(* CODESYS project wagolib787_01_twincat.library
   Company: Wago
   Title: T3_WagoLib787_01_TwinCat
   Placeholder: T3_WagoLib787_01_TwinCat
   Version: 1.0.0.0

Project tree, tasks and I/O mapping:
  libraries: Tc2_Standard, * (Beckhoff Automation GmbH); Tc2_System, * (Beckhoff Automation GmbH); Tc3_Interfaces, * (Beckhoff Automation GmbH); Tc3_Module, * (Beckhoff Automation GmbH)
  Data types/
    data type typEpsitronStatus
  Global Variables/
    global variables Global_Variables
    global variables Variable_Configuration
  POUs/
    function block FB787_1662 [ST]
    function block FB787_1662_ReadCurrent [ST]
    function block FB787_1664 [ST]
    function block FB787_1664_ReadCurrent [ST]
    function block FB787_1668 [ST]
    function block FB787_1668_ReadCurrent [ST]
    function FC787_Version [ST]
  Version/
    global variables Global_Version
  Visualizations/
*)

// Data types/typEpsitronStatus
TYPE typEpsitronStatus :
	(Ch_Active:=0,
	Ch_Warning:=1,
	Ch_Tripped:=2,
	Ch_not_Active:=3);
END_TYPE

// Global Variables/Global_Variables
{attribute 'Tc2GvlVarNames'}
VAR_GLOBAL
END_VAR

// Global Variables/Variable_Configuration
{attribute 'Tc2GvlVarNames'}
VAR_CONFIG
END_VAR

// Version/Global_Version
// This function has been automatically generated from the project information.
VAR_GLOBAL CONSTANT
	{attribute 'const_non_replaced'}
	{attribute 'linkalways'}
	stLibVersion_T3_WagoLib787_01_TwinCat : ST_LibVersion := (iMajor := 1, iMinor := 0, iBuild := 0, iRevision := 0, sVersion := '1.0.0.0');
END_VAR

// POUs/FB787_1662
FUNCTION_BLOCK FB787_1662
(***********************************************************************************************************	*)
(* Version: 1.0                                    			          														*)
(* Date: 05.09.2013                                   					          							            			*)
(***********************************************************************************************************	*)
(* WAGO Kontakttechnik GmbH Hansastr. 27 32423 Minden(Westf.)									*)
(* Tel. +0049 571/887-0 Fax. +0049 571/887-0															*)
(* Author: VB																								*)
(***********************************************************************************************************	*)
(*Description:	Epsitron electronic fuse (2 channel)	 													*)
(*Historie:																									*)
(*05.09.2013	VB		 Release																			*)
(***********************************************************************************************************	*)
VAR_INPUT
	xActive							:BOOL;
	xConfig						:BOOL;
	xChannel1Active				:BOOL;
	xChannel2Active				:BOOL;
	xS2_Input						:BOOL;
END_VAR
VAR_OUTPUT
	xDone							:BOOL;
	xConfigBusy					:BOOL;
	typChannel1Status			:typEpsitronStatus;(*0:Active,1:Warning,2:Tripped*)
	typChannel2Status			:typEpsitronStatus;
	xS1_Output					:BOOL;
END_VAR
VAR_IN_OUT
	xReset							:BOOL;
END_VAR
VAR
	a								: INT;
	state							: INT;
	TON1							: TON;
	aDaten						: ARRAY[0..44] OF BOOL;
	i								: INT;
	Ausgabe						: ARRAY[0..40] OF BOOL;
	go								: BOOL;
	init								: BOOL;
	R_TRIG1						: R_TRIG;
	auxExecute					: BOOL;
	xChannel3Active				:BOOL;
	xChannel4Active				:BOOL;
	xChannel5Active				: BOOL;
	xChannel6Active				: BOOL;
	xChannel7Active				: BOOL;
	xChannel8Active				: BOOL;
	auxReset						: BOOL;
END_VAR

IF xActive THEN
	R_TRIG1(CLK:=xConfig);
	IF r_trig1.q THEN
		auxExecute:=TRUE;
	END_IF
	
	CASE state OF
	0:(*ca. 1 Sekunde warten bis der Status abgefragt wird*)

		xS1_Output:=FALSE;
	
		IF NOT init THEN
			Ausgabe[0]:=1;
			Ausgabe[1]:=0;
			Ausgabe[2]:=1;
			Ausgabe[3]:=0;
			Ausgabe[4]:=1;
			Ausgabe[5]:=0;
			Ausgabe[6]:=1;
			Ausgabe[7]:=0;
			Ausgabe[8]:=1;
			Ausgabe[9]:=0;
			Ausgabe[10]:=1;
			Ausgabe[11]:=0;
			Ausgabe[12]:=1;
			Ausgabe[13]:=0;
			Ausgabe[14]:=1;
			Ausgabe[15]:=0;
			Ausgabe[16]:=1;
			Ausgabe[17]:=0;
			Ausgabe[18]:=1;
			Ausgabe[19]:=0;
			Ausgabe[20]:=1;
			Ausgabe[21]:=0;
			Ausgabe[22]:=1;
			Ausgabe[23]:=0;
			Ausgabe[24]:=1;
			Ausgabe[25]:=0;
			Ausgabe[26]:=1;
			Ausgabe[27]:=0;
			Ausgabe[28]:=1;
			Ausgabe[29]:=0;
			Ausgabe[30]:=1;
			Ausgabe[31]:=0;
			Ausgabe[32]:=1;
			Ausgabe[33]:=0;
			Ausgabe[34]:=0;
			Ausgabe[35]:=0;
			Ausgabe[36]:=0;
			Ausgabe[37]:=0;
			Ausgabe[38]:=0;
			Ausgabe[39]:=0;
			Ausgabe[40]:=0;
			init:=TRUE;
		END_IF

		IF auxExecute  THEN
			xConfigBusy:=TRUE;
			go:=TRUE;
			Ausgabe[0]:=1;
			Ausgabe[1]:=0;
			IF xChannel8Active THEN
				Ausgabe[2]:=0;
				Ausgabe[3]:=1;
			ELSE
				Ausgabe[2]:=1;
				Ausgabe[3]:=0;
			END_IF
		
			IF xChannel7Active THEN
				Ausgabe[4]:=0;
				Ausgabe[5]:=1;
			ELSE
				Ausgabe[4]:=1;
				Ausgabe[5]:=0;
			END_IF
			IF xChannel6Active THEN
				Ausgabe[6]:=0;
				Ausgabe[7]:=1;
			ELSE
				Ausgabe[6]:=1;
				Ausgabe[7]:=0;
			END_IF
			IF xChannel5Active THEN
				Ausgabe[8]:=0;
				Ausgabe[9]:=1;
			ELSE
				Ausgabe[8]:=1;
				Ausgabe[9]:=0;
			END_IF
			IF xChannel4Active THEN
				Ausgabe[10]:=0;
				Ausgabe[11]:=1;
			ELSE
				Ausgabe[10]:=1;
				Ausgabe[11]:=0;
			END_IF
			IF xChannel3Active THEN
				Ausgabe[12]:=0;
				Ausgabe[13]:=1;
			ELSE
				Ausgabe[12]:=1;
				Ausgabe[13]:=0;
			END_IF
			IF xChannel2Active THEN
				Ausgabe[14]:=0;
				Ausgabe[15]:=1;
			ELSE
				Ausgabe[14]:=1;
				Ausgabe[15]:=0;
			END_IF
			IF xChannel1Active THEN
				Ausgabe[16]:=0;
				Ausgabe[17]:=1;
			ELSE
				Ausgabe[16]:=1;
				Ausgabe[17]:=0;
			END_IF
			IF go THEN
				Ausgabe[18]:=0;
				Ausgabe[19]:=1;
			ELSE
				Ausgabe[18]:=1;
				Ausgabe[19]:=0;
			END_IF
				Ausgabe[20]:=1;
				Ausgabe[21]:=0;
				Ausgabe[22]:=1;
				Ausgabe[23]:=0;
				Ausgabe[24]:=1;
				Ausgabe[25]:=0;
				Ausgabe[26]:=1;
				Ausgabe[27]:=0;
				Ausgabe[28]:=1;
				Ausgabe[29]:=0;
				Ausgabe[30]:=1;
				Ausgabe[31]:=0;
				Ausgabe[32]:=1;
				Ausgabe[33]:=0;
				Ausgabe[34]:=0;
				Ausgabe[35]:=0;
				Ausgabe[36]:=0;
				Ausgabe[37]:=0;
				Ausgabe[38]:=0;
				Ausgabe[39]:=0;
				Ausgabe[40]:=0;
		END_IF;
	
		TON1(IN:=TRUE , PT:=t#1s);
		IF ton1.Q THEN
			state:=3;
			TON1(IN:=FALSE);
		END_IF


		(*Channel 1*)
		IF (aDaten[34] AND aDaten[35]) AND (aDaten[18] AND aDaten[19]) THEN
			typChannel1Status:=1;
		ELSIF (aDaten[34] AND aDaten[35]) AND (aDaten[18]=FALSE AND aDaten[19]=FALSE) THEN
			typChannel1Status:=2;
		ELSIF (aDaten[34]=FALSE AND aDaten[35]=FALSE) AND (aDaten[18]=FALSE AND aDaten[19]=FALSE) THEN
			typChannel1Status:=3;
		ELSE
			typChannel1Status:=0;
		END_IF

		(*Channel 2*)
		IF (aDaten[32] AND aDaten[33]) AND (aDaten[16] AND aDaten[17]) THEN
			typChannel2Status:=1;
		ELSIF (aDaten[32] AND aDaten[33]) AND (aDaten[16]=FALSE AND aDaten[17]=FALSE) THEN
			typChannel2Status:=2;
		ELSIF (aDaten[32]=FALSE AND aDaten[33]=FALSE) AND (aDaten[16]=FALSE AND aDaten[17]=FALSE) THEN
			typChannel2Status:=3;
		ELSE
			typChannel2Status:=0;
		END_IF


		IF auxReset AND xReset THEN
			xReset:=FALSE;
			auxReset:=FALSE;
		END_IF

	3:(*Reset Impuls mit 500ms ausführen*)
		IF xReset  THEN
			xS1_Output:=TRUE;
			TON1(IN:=TRUE , PT:=t#500ms);
			IF ton1.Q THEN
				state:=4;
				TON1(IN:=FALSE);
			END_IF
		ELSE
			state:=5;
			xS1_Output:=FALSE;
		END_IF
	
	4:(*Pause nach Reset*)
		TON1(IN:=TRUE , PT:=t#300ms);
		xS1_Output:=FALSE;
		IF ton1.Q THEN
			state:=5;
			TON1(IN:=FALSE);
			auxReset:=TRUE;
		END_IF

	5:
	(*Daten anfragen*)

		xS1_Output:=Ausgabe[a];
		aDaten[a+1]:=xS2_Input;
		a:=a+1;

		IF a>40 THEN
			state:=0;
			a:=0;
			i:=0;
			go:=FALSE;
			IF 	auxExecute AND xConfigBusy THEN(*schreibauftrag erledigt*)
				xDone:=FALSE;
				auxExecute:=FALSE;
				init:=FALSE;(*damit anschließend nur Daten ausgelesen werden. muss das Feld wieder den Lesecode bekommen*)
			ELSIF auxExecute AND NOT xConfigBusy THEN(*neuer  Schreibauftrag eingetroffen*)
				xConfigBusy:=TRUE;
				xDone:=FALSE;
			ELSE
				IF xConfig THEN
					xDone:=TRUE;
				ELSE
					xDone:=FALSE;
				END_IF
				xConfigBusy:=FALSE;
			END_IF
		ELSE
			;
		END_IF

	END_CASE
ELSE
	xS1_Output:=FALSE;
	state:=0;
	init:=0;
	a:=0;
	i:=0;
	auxReset:=FALSE;
END_IF

END_FUNCTION_BLOCK

// POUs/FB787_1662_ReadCurrent
FUNCTION_BLOCK FB787_1662_ReadCurrent
(***********************************************************************************************************	*)
(* Version: 1.0                                    			          														*)
(* Date: 05.09.2013                                   					          							            			*)
(***********************************************************************************************************	*)
(* WAGO Kontakttechnik GmbH Hansastr. 27 32423 Minden(Westf.)									*)
(* Tel. +0049 571/887-0 Fax. +0049 571/887-0															*)
(* Author: VB																								*)
(***********************************************************************************************************	*)
(*Description:	Epsitron electronic fuse with current overload protection	 							*)
(*Historie:																									*)
(*05.09.2013	VB		 			  																		*)
(***********************************************************************************************************	*)
VAR_INPUT
	xActive							:BOOL;
	xConfig						:BOOL;
	xChannel1Active				:BOOL;
	xChannel2Active				:BOOL;
	xReadSetting					:BOOL;(*0:read current,1:read setting*)
	xS2_Input						:BOOL;
END_VAR
VAR_OUTPUT
	xDone							:BOOL;
	xConfigBusy					:BOOL;
	typChannel1Status			:typEpsitronStatus;(*0:active,1:Überlast,2:Tripped,3:not_active*)
	typChannel2Status			:typEpsitronStatus;
	rVoltage						:REAL;
	rChannel1Current				:REAL;
	rChannel2Current				:REAL;
	iauxDisplay					:INT;
	xDisplaySettings				:BOOL;(*0:Channel value is current, 1:Channel value is setting*)
	xS1_Output					:BOOL;
END_VAR
VAR_IN_OUT
	xReset							:BOOL;
END_VAR
VAR
	xChannel3Active				:BOOL;
	xChannel4Active				:BOOL;
	xChannel5Active				:BOOL;
	xChannel6Active				:BOOL;
	xChannel7Active				:BOOL;
	xChannel8Active				:BOOL;
	typChannel3Status			:typEpsitronStatus;
	typChannel4Status			:typEpsitronStatus;
	typChannel5Status			:typEpsitronStatus;
	typChannel6Status			:typEpsitronStatus;
	typChannel7Status			:typEpsitronStatus;
	typChannel8Status			:typEpsitronStatus;
	rChannel3Current				:REAL;
	rChannel4Current				:REAL;
	rChannel5Current				:REAL;
	rChannel6Current				:REAL;
	rChannel7Current				:REAL;
	rChannel8Current				:REAL;
	a								: INT;
	state							: INT;
	TON1							: TON;
	aDaten						: ARRAY[0..188] OF BOOL;
	i								: INT;
	Ausgabe						: ARRAY[0..188] OF BOOL;
	go								: BOOL;
	init								: BOOL;
	R_TRIG1						: R_TRIG;
	auxExecute					: BOOL;
	auxReset						: BOOL;
	k								: INT;
	m								: INT;
	auxbyte						: BYTE;
	accurrentaux					: ARRAY[0..7]OF BYTE;
	bVoltage						: BYTE;
	auxProtocolBit5				: BOOL;
END_VAR

IF xActive THEN
	R_TRIG1(CLK:=xConfig);
	IF r_trig1.q THEN
		auxExecute:=TRUE;
	END_IF
	
	CASE state OF
	0:(*ca. 1 Sekunde warten bis der Status abgefragt wird*)

		xS1_Output:=FALSE;

		IF xReadSetting THEN
			Ausgabe[22]:=0;(*Bit 5->true*)
			Ausgabe[23]:=1;
		ELSE
			Ausgabe[22]:=1;
			Ausgabe[23]:=0;
		END_IF

		IF NOT init THEN
			FOR k:=0 TO 89 DO
				Ausgabe[2*k]:=1;
				Ausgabe[2*k+1]:=0;
			END_FOR
			FOR k:=0 TO 8 DO
				Ausgabe[178+k]:=0;
			END_FOR
			(*Protokoll 89 Bit*)
			Ausgabe[20]:=0;(*bit 6->true*)
			Ausgabe[21]:=1;

			IF xReadSetting THEN
				Ausgabe[22]:=0;(*Bit 5->true*)
				Ausgabe[23]:=1;
			ELSE
				Ausgabe[22]:=1;
				Ausgabe[23]:=0;
			END_IF

			init:=TRUE;
		END_IF

		IF auxExecute  THEN
			xConfigBusy:=TRUE;
			go:=TRUE;
			Ausgabe[0]:=1;
			Ausgabe[1]:=0;
			IF xChannel8Active THEN
				Ausgabe[2]:=0;
				Ausgabe[3]:=1;
			ELSE
				Ausgabe[2]:=1;
				Ausgabe[3]:=0;
			END_IF
		
			IF xChannel7Active THEN
				Ausgabe[4]:=0;
				Ausgabe[5]:=1;
			ELSE
				Ausgabe[4]:=1;
				Ausgabe[5]:=0;
			END_IF
			IF xChannel6Active THEN
				Ausgabe[6]:=0;
				Ausgabe[7]:=1;
			ELSE
				Ausgabe[6]:=1;
				Ausgabe[7]:=0;
			END_IF
			IF xChannel5Active THEN
				Ausgabe[8]:=0;
				Ausgabe[9]:=1;
			ELSE
				Ausgabe[8]:=1;
				Ausgabe[9]:=0;
			END_IF
			IF xChannel4Active THEN
				Ausgabe[10]:=0;
				Ausgabe[11]:=1;
			ELSE
				Ausgabe[10]:=1;
				Ausgabe[11]:=0;
			END_IF
			IF xChannel3Active THEN
				Ausgabe[12]:=0;
				Ausgabe[13]:=1;
			ELSE
				Ausgabe[12]:=1;
				Ausgabe[13]:=0;
			END_IF
			IF xChannel2Active THEN
				Ausgabe[14]:=0;
				Ausgabe[15]:=1;
			ELSE
				Ausgabe[14]:=1;
				Ausgabe[15]:=0;
			END_IF
			IF xChannel1Active THEN
				Ausgabe[16]:=0;
				Ausgabe[17]:=1;
			ELSE
				Ausgabe[16]:=1;
				Ausgabe[17]:=0;
			END_IF
			IF go THEN
				Ausgabe[18]:=0;
				Ausgabe[19]:=1;
			ELSE
				Ausgabe[18]:=1;
				Ausgabe[19]:=0;
			END_IF
			(*Protokoll 89 Bit*)
			Ausgabe[20]:=0;
			Ausgabe[21]:=1;
			IF xReadSetting THEN
				Ausgabe[22]:=0;(*Bit 5->true*)
				Ausgabe[23]:=1;
			ELSE
				Ausgabe[22]:=1;
				Ausgabe[23]:=0;
			END_IF

				FOR k:=0 TO 79 DO
					Ausgabe[24+2*k]:=1;
					Ausgabe[25+2*k]:=0;
				END_FOR

				Ausgabe[178]:=0;
				Ausgabe[179]:=0;
				Ausgabe[180]:=0;
				Ausgabe[181]:=0;
				Ausgabe[182]:=0;
				Ausgabe[183]:=0;
				Ausgabe[184]:=0;
				Ausgabe[185]:=0;
				Ausgabe[186]:=0;
				Ausgabe[187]:=0;
				Ausgabe[188]:=0;

		END_IF;

		TON1(IN:=TRUE , PT:=t#1s);
		IF ton1.Q THEN
			state:=3;
			TON1(IN:=FALSE);
		END_IF


		(*Channel 1*)
		IF (aDaten[34] (*AND aDaten[35]*)) AND (aDaten[18] AND aDaten[19]) THEN
			typChannel1Status:=1;
		ELSIF (aDaten[34] (*AND aDaten[35]*)) AND (aDaten[18]=FALSE AND aDaten[19]=FALSE) THEN
			typChannel1Status:=2;
		ELSIF (aDaten[34]=FALSE AND aDaten[35]=FALSE) AND (aDaten[18]=FALSE AND aDaten[19]=FALSE) THEN
			typChannel1Status:=3;
		ELSE
			typChannel1Status:=0;
		END_IF

		(*Channel 2*)
		IF (aDaten[32] AND aDaten[33]) AND (aDaten[16] AND aDaten[17]) THEN
			typChannel2Status:=1;
		ELSIF (aDaten[32] AND aDaten[33]) AND (aDaten[16]=FALSE AND aDaten[17]=FALSE) THEN
			typChannel2Status:=2;
		ELSIF (aDaten[32]=FALSE AND aDaten[33]=FALSE) AND (aDaten[16]=FALSE AND aDaten[17]=FALSE) THEN
			typChannel2Status:=3;
		ELSE
			typChannel2Status:=0;
		END_IF

		(*Channel 3*)
		IF (aDaten[30] AND aDaten[31]) AND (aDaten[14] AND aDaten[15]) THEN
			typChannel3Status:=1;
		ELSIF (aDaten[30] AND aDaten[31]) AND (aDaten[14]=FALSE AND aDaten[15]=FALSE) THEN
			typChannel3Status:=2;
		ELSIF (aDaten[30]=FALSE AND aDaten[31]=FALSE) AND (aDaten[14]=FALSE AND aDaten[15]=FALSE) THEN
			typChannel3Status:=3;
		ELSE
			typChannel3Status:=0;
		END_IF

		(*Channel 4*)
		IF (aDaten[28] AND aDaten[29]) AND (aDaten[12] AND aDaten[13]) THEN
			typChannel4Status:=1;
		ELSIF (aDaten[28] AND aDaten[29]) AND (aDaten[12]=FALSE AND aDaten[13]=FALSE) THEN
			typChannel4Status:=2;
		ELSIF (aDaten[28]=FALSE AND aDaten[29]=FALSE) AND (aDaten[12]=FALSE AND aDaten[13]=FALSE) THEN
			typChannel4Status:=3;
		ELSE
			typChannel4Status:=0;
		END_IF

	(*Channel 5*)
		IF (aDaten[26] AND aDaten[27]) AND (aDaten[10] AND aDaten[11]) THEN
			typChannel5Status:=1;
		ELSIF (aDaten[26] AND aDaten[27]) AND (aDaten[10]=FALSE AND aDaten[11]=FALSE) THEN
			typChannel5Status:=2;
		ELSIF (aDaten[26]=FALSE AND aDaten[27]=FALSE) AND (aDaten[10]=FALSE AND aDaten[11]=FALSE) THEN
			typChannel5Status:=3;
		ELSE
			typChannel5Status:=0;
		END_IF

	(*Channel 6*)
		IF (aDaten[24] AND aDaten[25]) AND (aDaten[8] AND aDaten[9]) THEN
			typChannel6Status:=1;
		ELSIF (aDaten[24] AND aDaten[25]) AND (aDaten[8]=FALSE AND aDaten[9]=FALSE) THEN
			typChannel6Status:=2;
		ELSIF (aDaten[24]=FALSE AND aDaten[25]=FALSE) AND (aDaten[8]=FALSE AND aDaten[9]=FALSE) THEN
			typChannel6Status:=3;
		ELSE
			typChannel6Status:=0;
		END_IF

	(*Channel 7*)
		IF (aDaten[22] AND aDaten[23]) AND (aDaten[6] AND aDaten[7]) THEN
			typChannel7Status:=1;
		ELSIF (aDaten[22] AND aDaten[23]) AND (aDaten[6]=FALSE AND aDaten[7]=FALSE) THEN
			typChannel7Status:=2;
		ELSIF (aDaten[22]=FALSE AND aDaten[23]=FALSE) AND (aDaten[6]=FALSE AND aDaten[7]=FALSE) THEN
			typChannel7Status:=3;
		ELSE
			typChannel7Status:=0;
		END_IF

	(*Channel 8*)
		IF (aDaten[20] AND aDaten[21]) AND (aDaten[4] AND aDaten[5]) THEN
			typChannel8Status:=1;
		ELSIF (aDaten[20] AND aDaten[21]) AND (aDaten[4]=FALSE AND aDaten[5]=FALSE) THEN
			typChannel8Status:=2;
		ELSIF (aDaten[20]=FALSE AND aDaten[21]=FALSE) AND (aDaten[4]=FALSE AND aDaten[5]=FALSE) THEN
			typChannel8Status:=3;
		ELSE
			typChannel8Status:=0;
		END_IF

		(*analog Werte Protokoll 89 bit*)
		IF (aDaten[36] AND aDaten[37]) THEN
			bVoltage.7:=TRUE;
		ELSE
			bVoltage.7:=FALSE;
		END_IF
		IF (aDaten[38] AND aDaten[39]) THEN
			bVoltage.6:=TRUE;
		ELSE
			bVoltage.6:=FALSE;
		END_IF
		IF (aDaten[40] AND aDaten[41]) THEN
			bVoltage.5:=TRUE;
		ELSE
			bVoltage.5:=FALSE;
		END_IF
		IF (aDaten[42] AND aDaten[43]) THEN
			bVoltage.4:=TRUE;
		ELSE
			bVoltage.4:=FALSE;
		END_IF
		IF (aDaten[44] AND aDaten[45]) THEN
			bVoltage.3:=TRUE;
		ELSE
			bVoltage.3:=FALSE;
		END_IF
		IF (aDaten[46] AND aDaten[47]) THEN
			bVoltage.2:=TRUE;
		ELSE
			bVoltage.2:=FALSE;
		END_IF
		IF (aDaten[48] AND aDaten[49]) THEN
			bVoltage.1:=TRUE;
		ELSE
			bVoltage.1:=FALSE;
		END_IF
		IF (aDaten[50] AND aDaten[51]) THEN
			bVoltage.0:=TRUE;
		ELSE
			bVoltage.0:=FALSE;
		END_IF
		IF bVoltage>0 THEN
			rVoltage:=BYTE_TO_REAL(bVoltage)/16+16;
		ELSE
			rVoltage:=0;
		END_IF

		FOR m:=0 TO 7 DO
			IF (aDaten[52+16*m] AND aDaten[53+16*m]) THEN
				auxbyte.7:=TRUE;
			ELSE
				auxbyte.7:=FALSE;
			END_IF
			IF (aDaten[54+16*m] AND aDaten[55+16*m]) THEN
				auxbyte.6:=TRUE;
			ELSE
				auxbyte.6:=FALSE;
			END_IF
			IF (aDaten[56+16*m] AND aDaten[57+16*m]) THEN
				auxbyte.5:=TRUE;
			ELSE
				auxbyte.5:=FALSE;
			END_IF
			IF (aDaten[58+16*m] AND aDaten[59+16*m]) THEN
				auxbyte.4:=TRUE;
			ELSE
				auxbyte.4:=FALSE;
			END_IF
			IF (aDaten[60+16*m] AND aDaten[61+16*m]) THEN
				auxbyte.3:=TRUE;
			ELSE
				auxbyte.3:=FALSE;
			END_IF
			IF (aDaten[62+16*m] AND aDaten[63+16*m]) THEN
				auxbyte.2:=TRUE;
			ELSE
				auxbyte.2:=FALSE;
			END_IF
			IF (aDaten[64+16*m] AND aDaten[65+16*m]) THEN
				auxbyte.1:=TRUE;
			ELSE
				auxbyte.1:=FALSE;
			END_IF
			IF (aDaten[66+16*m] AND aDaten[67+16*m]) THEN
				auxbyte.0:=TRUE;
			ELSE
				auxbyte.0:=FALSE;
			END_IF
			accurrentaux[m]:=auxbyte;
		END_FOR
		rChannel1Current:=BYTE_TO_REAL(accurrentaux[0])/16;
		rChannel2Current:=BYTE_TO_REAL(accurrentaux[1])/16;
		rChannel3Current:=BYTE_TO_REAL(accurrentaux[2])/16;
		rChannel4Current:=BYTE_TO_REAL(accurrentaux[3])/16;
		rChannel5Current:=BYTE_TO_REAL(accurrentaux[4])/16;
		rChannel6Current:=BYTE_TO_REAL(accurrentaux[5])/16;
		rChannel7Current:=BYTE_TO_REAL(accurrentaux[6])/16;
		rChannel8Current:=BYTE_TO_REAL(accurrentaux[7])/16;

		(*indicates wether current or setting values are displayed*)
		xDisplaySettings:=auxProtocolBit5;

		IF auxReset AND xReset THEN
			xReset:=FALSE;
			auxReset:=FALSE;
		END_IF

	3:(*Reset Impuls mit 500ms ausführen*)
		IF xReset  THEN
			xS1_Output:=TRUE;
			TON1(IN:=TRUE , PT:=t#500ms);
			IF ton1.Q THEN
				state:=4;
				TON1(IN:=FALSE);
			END_IF
		ELSE
			state:=5;
			xS1_Output:=FALSE;
		END_IF

	4:(*Pause nach Reset*)
		TON1(IN:=TRUE , PT:=t#300ms);
		xS1_Output:=FALSE;
		IF ton1.Q THEN
			state:=5;
			TON1(IN:=FALSE);
			auxReset:=TRUE;
		END_IF

	5:
	(*Daten anfragen*)

		xS1_Output:=Ausgabe[a];
		aDaten[a+1]:=xS2_Input;
		a:=a+1;
		iauxDisplay:=a;
		auxProtocolBit5:=NOT Ausgabe[22]; (*remember which values should be displayed->current or setting, dependen on bit5*)
		(*IF a>40 THEN*)
		IF a>184 THEN
			state:=0;
			a:=0;
			i:=0;
			go:=FALSE;
			IF 	auxExecute AND xConfigBusy THEN(*schreibauftrag erledigt*)
				xDone:=FALSE;
				auxExecute:=FALSE;
				init:=FALSE;(*damit anschließend nur Daten ausgelesen werden. muss das Feld wieder den Lesecode bekommen*)
			ELSIF auxExecute AND NOT xConfigBusy THEN(*neuer  Schreibauftrag eingetroffen*)
				xConfigBusy:=TRUE;
				xDone:=FALSE;
			ELSE
				IF xConfig THEN
					xDone:=TRUE;
				ELSE
					xDone:=FALSE;
				END_IF
				xConfigBusy:=FALSE;
			END_IF
		ELSE
			;
		END_IF

	END_CASE
ELSE
	xS1_Output:=FALSE;
	state:=0;
	init:=0;
	a:=0;
	i:=0;
	auxReset:=FALSE;
END_IF

END_FUNCTION_BLOCK

// POUs/FB787_1664
FUNCTION_BLOCK FB787_1664
(***********************************************************************************************************	*)
(* Version: 0.8                                    			          														*)
(* Date: 01.07.2012                                   					          							            			*)
(***********************************************************************************************************	*)
(* WAGO Kontakttechnik GmbH Hansastr. 27 32423 Minden(Westf.)									*)
(* Tel. +0049 571/887-0 Fax. +0049 571/887-0															*)
(* Author: VB																								*)
(***********************************************************************************************************	*)
(*Description:	Epsitron electronic fuse	 																*)
(*Historie:																									*)
(*01.07.2013	VB		 Version 0.8 changes according to FW2.00										*)
(*22.10.2012	VB		 Version 0.7 RC																	*)
(***********************************************************************************************************	*)
VAR_INPUT
	xActive							:BOOL;
	xConfig						:BOOL;
	xChannel1Active				:BOOL;
	xChannel2Active				:BOOL;
	xChannel3Active				:BOOL;
	xChannel4Active				:BOOL;
	xS2_Input						:BOOL;
END_VAR
VAR_OUTPUT
	xDone							:BOOL;
	xConfigBusy					:BOOL;
	typChannel1Status			:typEpsitronStatus;(*0:Active,1:Warning,2:Tripped*)
	typChannel2Status			:typEpsitronStatus;
	typChannel3Status			:typEpsitronStatus;
	typChannel4Status			:typEpsitronStatus;
	xS1_Output					:BOOL;
END_VAR
VAR_IN_OUT
	xReset							:BOOL;
END_VAR
VAR
	a								: INT;
	state							: INT;
	TON1							: TON;
	aDaten						: ARRAY[0..44] OF BOOL;
	i								: INT;
	Ausgabe						: ARRAY[0..40] OF BOOL;
	go								: BOOL;
	init								: BOOL;
	R_TRIG1						: R_TRIG;
	auxExecute					: BOOL;
	xChannel5Active				: BOOL;
	xChannel6Active				: BOOL;
	xChannel7Active				: BOOL;
	xChannel8Active				: BOOL;
	auxReset						: BOOL;
END_VAR

IF xActive THEN
	R_TRIG1(CLK:=xConfig);
	IF r_trig1.q THEN
		auxExecute:=TRUE;
	END_IF
	
	CASE state OF
	0:(*ca. 1 Sekunde warten bis der Status abgefragt wird*)

		xS1_Output:=FALSE;
	
		IF NOT init THEN
			Ausgabe[0]:=1;
			Ausgabe[1]:=0;
			Ausgabe[2]:=1;
			Ausgabe[3]:=0;
			Ausgabe[4]:=1;
			Ausgabe[5]:=0;
			Ausgabe[6]:=1;
			Ausgabe[7]:=0;
			Ausgabe[8]:=1;
			Ausgabe[9]:=0;
			Ausgabe[10]:=1;
			Ausgabe[11]:=0;
			Ausgabe[12]:=1;
			Ausgabe[13]:=0;
			Ausgabe[14]:=1;
			Ausgabe[15]:=0;
			Ausgabe[16]:=1;
			Ausgabe[17]:=0;
			Ausgabe[18]:=1;
			Ausgabe[19]:=0;
			Ausgabe[20]:=1;
			Ausgabe[21]:=0;
			Ausgabe[22]:=1;
			Ausgabe[23]:=0;
			Ausgabe[24]:=1;
			Ausgabe[25]:=0;
			Ausgabe[26]:=1;
			Ausgabe[27]:=0;
			Ausgabe[28]:=1;
			Ausgabe[29]:=0;
			Ausgabe[30]:=1;
			Ausgabe[31]:=0;
			Ausgabe[32]:=1;
			Ausgabe[33]:=0;
			Ausgabe[34]:=0;
			Ausgabe[35]:=0;
			Ausgabe[36]:=0;
			Ausgabe[37]:=0;
			Ausgabe[38]:=0;
			Ausgabe[39]:=0;
			Ausgabe[40]:=0;
			init:=TRUE;
		END_IF

		IF auxExecute  THEN
			xConfigBusy:=TRUE;
			go:=TRUE;
			Ausgabe[0]:=1;
			Ausgabe[1]:=0;
			IF xChannel8Active THEN
				Ausgabe[2]:=0;
				Ausgabe[3]:=1;
			ELSE
				Ausgabe[2]:=1;
				Ausgabe[3]:=0;
			END_IF
		
			IF xChannel7Active THEN
				Ausgabe[4]:=0;
				Ausgabe[5]:=1;
			ELSE
				Ausgabe[4]:=1;
				Ausgabe[5]:=0;
			END_IF
			IF xChannel6Active THEN
				Ausgabe[6]:=0;
				Ausgabe[7]:=1;
			ELSE
				Ausgabe[6]:=1;
				Ausgabe[7]:=0;
			END_IF
			IF xChannel5Active THEN
				Ausgabe[8]:=0;
				Ausgabe[9]:=1;
			ELSE
				Ausgabe[8]:=1;
				Ausgabe[9]:=0;
			END_IF
			IF xChannel4Active THEN
				Ausgabe[10]:=0;
				Ausgabe[11]:=1;
			ELSE
				Ausgabe[10]:=1;
				Ausgabe[11]:=0;
			END_IF
			IF xChannel3Active THEN
				Ausgabe[12]:=0;
				Ausgabe[13]:=1;
			ELSE
				Ausgabe[12]:=1;
				Ausgabe[13]:=0;
			END_IF
			IF xChannel2Active THEN
				Ausgabe[14]:=0;
				Ausgabe[15]:=1;
			ELSE
				Ausgabe[14]:=1;
				Ausgabe[15]:=0;
			END_IF
			IF xChannel1Active THEN
				Ausgabe[16]:=0;
				Ausgabe[17]:=1;
			ELSE
				Ausgabe[16]:=1;
				Ausgabe[17]:=0;
			END_IF
			IF go THEN
				Ausgabe[18]:=0;
				Ausgabe[19]:=1;
			ELSE
				Ausgabe[18]:=1;
				Ausgabe[19]:=0;
			END_IF
				Ausgabe[20]:=1;
				Ausgabe[21]:=0;
				Ausgabe[22]:=1;
				Ausgabe[23]:=0;
				Ausgabe[24]:=1;
				Ausgabe[25]:=0;
				Ausgabe[26]:=1;
				Ausgabe[27]:=0;
				Ausgabe[28]:=1;
				Ausgabe[29]:=0;
				Ausgabe[30]:=1;
				Ausgabe[31]:=0;
				Ausgabe[32]:=1;
				Ausgabe[33]:=0;
				Ausgabe[34]:=0;
				Ausgabe[35]:=0;
				Ausgabe[36]:=0;
				Ausgabe[37]:=0;
				Ausgabe[38]:=0;
				Ausgabe[39]:=0;
				Ausgabe[40]:=0;
		END_IF;
	
		TON1(IN:=TRUE , PT:=t#1s);
		IF ton1.Q THEN
			state:=3;
			TON1(IN:=FALSE);
		END_IF


		(*Channel 1*)
		IF (aDaten[34] AND aDaten[35]) AND (aDaten[18] AND aDaten[19]) THEN
			typChannel1Status:=1;
		ELSIF (aDaten[34] AND aDaten[35]) AND (aDaten[18]=FALSE AND aDaten[19]=FALSE) THEN
			typChannel1Status:=2;
		ELSIF (aDaten[34]=FALSE AND aDaten[35]=FALSE) AND (aDaten[18]=FALSE AND aDaten[19]=FALSE) THEN
			typChannel1Status:=3;
		ELSE
			typChannel1Status:=0;
		END_IF

		(*Channel 2*)
		IF (aDaten[32] AND aDaten[33]) AND (aDaten[16] AND aDaten[17]) THEN
			typChannel2Status:=1;
		ELSIF (aDaten[32] AND aDaten[33]) AND (aDaten[16]=FALSE AND aDaten[17]=FALSE) THEN
			typChannel2Status:=2;
		ELSIF (aDaten[32]=FALSE AND aDaten[33]=FALSE) AND (aDaten[16]=FALSE AND aDaten[17]=FALSE) THEN
			typChannel2Status:=3;
		ELSE
			typChannel2Status:=0;
		END_IF

		(*Channel 3*)
		IF (aDaten[30] AND aDaten[31]) AND (aDaten[14] AND aDaten[15]) THEN
			typChannel3Status:=1;
		ELSIF (aDaten[30] AND aDaten[31]) AND (aDaten[14]=FALSE AND aDaten[15]=FALSE) THEN
			typChannel3Status:=2;
		ELSIF (aDaten[30]=FALSE AND aDaten[31]=FALSE) AND (aDaten[14]=FALSE AND aDaten[15]=FALSE) THEN
			typChannel3Status:=3;
		ELSE
			typChannel3Status:=0;
		END_IF

		(*Channel 4*)
		IF (aDaten[28] AND aDaten[29]) AND (aDaten[12] AND aDaten[13]) THEN
			typChannel4Status:=1;
		ELSIF (aDaten[28] AND aDaten[29]) AND (aDaten[12]=FALSE AND aDaten[13]=FALSE) THEN
			typChannel4Status:=2;
		ELSIF (aDaten[28]=FALSE AND aDaten[29]=FALSE) AND (aDaten[12]=FALSE AND aDaten[13]=FALSE) THEN
			typChannel4Status:=3;
		ELSE
			typChannel4Status:=0;
		END_IF



		IF auxReset AND xReset THEN
			xReset:=FALSE;
			auxReset:=FALSE;
		END_IF

	3:(*Reset Impuls mit 500ms ausführen*)
		IF xReset  THEN
			xS1_Output:=TRUE;
			TON1(IN:=TRUE , PT:=t#500ms);
			IF ton1.Q THEN
				state:=4;
				TON1(IN:=FALSE);
			END_IF
		ELSE
			state:=5;
			xS1_Output:=FALSE;
		END_IF
	
	4:(*Pause nach Reset*)
		TON1(IN:=TRUE , PT:=t#300ms);
		xS1_Output:=FALSE;
		IF ton1.Q THEN
			state:=5;
			TON1(IN:=FALSE);
			auxReset:=TRUE;
		END_IF

	5:
	(*Daten anfragen*)

		xS1_Output:=Ausgabe[a];
		aDaten[a+1]:=xS2_Input;
		a:=a+1;

		IF a>40 THEN
			state:=0;
			a:=0;
			i:=0;
			go:=FALSE;
			IF 	auxExecute AND xConfigBusy THEN(*schreibauftrag erledigt*)
				xDone:=FALSE;
				auxExecute:=FALSE;
				init:=FALSE;(*damit anschließend nur Daten ausgelesen werden. muss das Feld wieder den Lesecode bekommen*)
			ELSIF auxExecute AND NOT xConfigBusy THEN(*neuer  Schreibauftrag eingetroffen*)
				xConfigBusy:=TRUE;
				xDone:=FALSE;
			ELSE
				IF xConfig THEN
					xDone:=TRUE;
				ELSE
					xDone:=FALSE;
				END_IF
				xConfigBusy:=FALSE;
			END_IF
		ELSE
			;
		END_IF

	END_CASE
ELSE
	xS1_Output:=FALSE;
	state:=0;
	init:=0;
	a:=0;
	i:=0;
	auxReset:=FALSE;
END_IF

END_FUNCTION_BLOCK

// POUs/FB787_1664_ReadCurrent
FUNCTION_BLOCK FB787_1664_ReadCurrent
(***********************************************************************************************************	*)
(* Version: 1.0                                    			          														*)
(* Date: 05.09.2013                                   					          							            			*)
(***********************************************************************************************************	*)
(* WAGO Kontakttechnik GmbH Hansastr. 27 32423 Minden(Westf.)									*)
(* Tel. +0049 571/887-0 Fax. +0049 571/887-0															*)
(* Author: VB																								*)
(***********************************************************************************************************	*)
(*Description:	Epsitron electronic fuse with current overload protection	 							*)
(*Historie:																									*)
(*05.09.2013	VB		 			released  																*)
(***********************************************************************************************************	*)
VAR_INPUT
	xActive							:BOOL;
	xConfig						:BOOL;
	xChannel1Active				:BOOL;
	xChannel2Active				:BOOL;
	xChannel3Active				:BOOL;
	xChannel4Active				:BOOL;
	xReadSetting					:BOOL;(*0:read current,1:read setting*)
	xS2_Input						:BOOL;
END_VAR
VAR_OUTPUT
	xDone							:BOOL;
	xConfigBusy					:BOOL;
	typChannel1Status			:typEpsitronStatus;(*0:active,1:Überlast,2:Tripped,3:not_active*)
	typChannel2Status			:typEpsitronStatus;
	typChannel3Status			:typEpsitronStatus;
	typChannel4Status			:typEpsitronStatus;
	rVoltage						:REAL;
	rChannel1Current				:REAL;
	rChannel2Current				:REAL;
	rChannel3Current				:REAL;
	rChannel4Current				:REAL;
	iauxDisplay					:INT;
	xDisplaySettings				:BOOL;(*0:Channel value is current, 1:Channel value is setting*)
	xS1_Output					:BOOL;
END_VAR
VAR_IN_OUT
	xReset							:BOOL;
END_VAR
VAR
	xChannel5Active				:BOOL;
	xChannel6Active				:BOOL;
	xChannel7Active				:BOOL;
	xChannel8Active				:BOOL;
	typChannel5Status			:typEpsitronStatus;
	typChannel6Status			:typEpsitronStatus;
	typChannel7Status			:typEpsitronStatus;
	typChannel8Status			:typEpsitronStatus;
	rChannel5Current				:REAL;
	rChannel6Current				:REAL;
	rChannel7Current				:REAL;
	rChannel8Current				:REAL;
	a								: INT;
	state							: INT;
	TON1							: TON;
	aDaten						: ARRAY[0..188] OF BOOL;
	i								: INT;
	Ausgabe						: ARRAY[0..188] OF BOOL;
	go								: BOOL;
	init								: BOOL;
	R_TRIG1						: R_TRIG;
	auxExecute					: BOOL;
	auxReset						: BOOL;
	k								: INT;
	m								: INT;
	auxbyte						: BYTE;
	accurrentaux					: ARRAY[0..7]OF BYTE;
	bVoltage						: BYTE;
	auxProtocolBit5				: BOOL;
END_VAR

IF xActive THEN
	R_TRIG1(CLK:=xConfig);
	IF r_trig1.q THEN
		auxExecute:=TRUE;
	END_IF
	
	CASE state OF
	0:(*ca. 1 Sekunde warten bis der Status abgefragt wird*)

		xS1_Output:=FALSE;

		IF xReadSetting THEN
			Ausgabe[22]:=0;(*Bit 5->true*)
			Ausgabe[23]:=1;
		ELSE
			Ausgabe[22]:=1;
			Ausgabe[23]:=0;
		END_IF

		IF NOT init THEN
			FOR k:=0 TO 89 DO
				Ausgabe[2*k]:=1;
				Ausgabe[2*k+1]:=0;
			END_FOR
			FOR k:=0 TO 8 DO
				Ausgabe[178+k]:=0;
			END_FOR
			(*Protokoll 89 Bit*)
			Ausgabe[20]:=0;(*bit 6->true*)
			Ausgabe[21]:=1;

			IF xReadSetting THEN
				Ausgabe[22]:=0;(*Bit 5->true*)
				Ausgabe[23]:=1;
			ELSE
				Ausgabe[22]:=1;
				Ausgabe[23]:=0;
			END_IF

			init:=TRUE;
		END_IF

		IF auxExecute  THEN
			xConfigBusy:=TRUE;
			go:=TRUE;
			Ausgabe[0]:=1;
			Ausgabe[1]:=0;
			IF xChannel8Active THEN
				Ausgabe[2]:=0;
				Ausgabe[3]:=1;
			ELSE
				Ausgabe[2]:=1;
				Ausgabe[3]:=0;
			END_IF
		
			IF xChannel7Active THEN
				Ausgabe[4]:=0;
				Ausgabe[5]:=1;
			ELSE
				Ausgabe[4]:=1;
				Ausgabe[5]:=0;
			END_IF
			IF xChannel6Active THEN
				Ausgabe[6]:=0;
				Ausgabe[7]:=1;
			ELSE
				Ausgabe[6]:=1;
				Ausgabe[7]:=0;
			END_IF
			IF xChannel5Active THEN
				Ausgabe[8]:=0;
				Ausgabe[9]:=1;
			ELSE
				Ausgabe[8]:=1;
				Ausgabe[9]:=0;
			END_IF
			IF xChannel4Active THEN
				Ausgabe[10]:=0;
				Ausgabe[11]:=1;
			ELSE
				Ausgabe[10]:=1;
				Ausgabe[11]:=0;
			END_IF
			IF xChannel3Active THEN
				Ausgabe[12]:=0;
				Ausgabe[13]:=1;
			ELSE
				Ausgabe[12]:=1;
				Ausgabe[13]:=0;
			END_IF
			IF xChannel2Active THEN
				Ausgabe[14]:=0;
				Ausgabe[15]:=1;
			ELSE
				Ausgabe[14]:=1;
				Ausgabe[15]:=0;
			END_IF
			IF xChannel1Active THEN
				Ausgabe[16]:=0;
				Ausgabe[17]:=1;
			ELSE
				Ausgabe[16]:=1;
				Ausgabe[17]:=0;
			END_IF
			IF go THEN
				Ausgabe[18]:=0;
				Ausgabe[19]:=1;
			ELSE
				Ausgabe[18]:=1;
				Ausgabe[19]:=0;
			END_IF
			(*Protokoll 89 Bit*)
			Ausgabe[20]:=0;
			Ausgabe[21]:=1;
			IF xReadSetting THEN
				Ausgabe[22]:=0;(*Bit 5->true*)
				Ausgabe[23]:=1;
			ELSE
				Ausgabe[22]:=1;
				Ausgabe[23]:=0;
			END_IF

				FOR k:=0 TO 79 DO
					Ausgabe[24+2*k]:=1;
					Ausgabe[25+2*k]:=0;
				END_FOR

				Ausgabe[178]:=0;
				Ausgabe[179]:=0;
				Ausgabe[180]:=0;
				Ausgabe[181]:=0;
				Ausgabe[182]:=0;
				Ausgabe[183]:=0;
				Ausgabe[184]:=0;
				Ausgabe[185]:=0;
				Ausgabe[186]:=0;
				Ausgabe[187]:=0;
				Ausgabe[188]:=0;

		END_IF;

		TON1(IN:=TRUE , PT:=t#1s);
		IF ton1.Q THEN
			state:=3;
			TON1(IN:=FALSE);
		END_IF


		(*Channel 1*)
		IF (aDaten[34] (*AND aDaten[35]*)) AND (aDaten[18] AND aDaten[19]) THEN
			typChannel1Status:=1;
		ELSIF (aDaten[34] (*AND aDaten[35]*)) AND (aDaten[18]=FALSE AND aDaten[19]=FALSE) THEN
			typChannel1Status:=2;
		ELSIF (aDaten[34]=FALSE AND aDaten[35]=FALSE) AND (aDaten[18]=FALSE AND aDaten[19]=FALSE) THEN
			typChannel1Status:=3;
		ELSE
			typChannel1Status:=0;
		END_IF

		(*Channel 2*)
		IF (aDaten[32] AND aDaten[33]) AND (aDaten[16] AND aDaten[17]) THEN
			typChannel2Status:=1;
		ELSIF (aDaten[32] AND aDaten[33]) AND (aDaten[16]=FALSE AND aDaten[17]=FALSE) THEN
			typChannel2Status:=2;
		ELSIF (aDaten[32]=FALSE AND aDaten[33]=FALSE) AND (aDaten[16]=FALSE AND aDaten[17]=FALSE) THEN
			typChannel2Status:=3;
		ELSE
			typChannel2Status:=0;
		END_IF

		(*Channel 3*)
		IF (aDaten[30] AND aDaten[31]) AND (aDaten[14] AND aDaten[15]) THEN
			typChannel3Status:=1;
		ELSIF (aDaten[30] AND aDaten[31]) AND (aDaten[14]=FALSE AND aDaten[15]=FALSE) THEN
			typChannel3Status:=2;
		ELSIF (aDaten[30]=FALSE AND aDaten[31]=FALSE) AND (aDaten[14]=FALSE AND aDaten[15]=FALSE) THEN
			typChannel3Status:=3;
		ELSE
			typChannel3Status:=0;
		END_IF

		(*Channel 4*)
		IF (aDaten[28] AND aDaten[29]) AND (aDaten[12] AND aDaten[13]) THEN
			typChannel4Status:=1;
		ELSIF (aDaten[28] AND aDaten[29]) AND (aDaten[12]=FALSE AND aDaten[13]=FALSE) THEN
			typChannel4Status:=2;
		ELSIF (aDaten[28]=FALSE AND aDaten[29]=FALSE) AND (aDaten[12]=FALSE AND aDaten[13]=FALSE) THEN
			typChannel4Status:=3;
		ELSE
			typChannel4Status:=0;
		END_IF

	(*Channel 5*)
		IF (aDaten[26] AND aDaten[27]) AND (aDaten[10] AND aDaten[11]) THEN
			typChannel5Status:=1;
		ELSIF (aDaten[26] AND aDaten[27]) AND (aDaten[10]=FALSE AND aDaten[11]=FALSE) THEN
			typChannel5Status:=2;
		ELSIF (aDaten[26]=FALSE AND aDaten[27]=FALSE) AND (aDaten[10]=FALSE AND aDaten[11]=FALSE) THEN
			typChannel5Status:=3;
		ELSE
			typChannel5Status:=0;
		END_IF

	(*Channel 6*)
		IF (aDaten[24] AND aDaten[25]) AND (aDaten[8] AND aDaten[9]) THEN
			typChannel6Status:=1;
		ELSIF (aDaten[24] AND aDaten[25]) AND (aDaten[8]=FALSE AND aDaten[9]=FALSE) THEN
			typChannel6Status:=2;
		ELSIF (aDaten[24]=FALSE AND aDaten[25]=FALSE) AND (aDaten[8]=FALSE AND aDaten[9]=FALSE) THEN
			typChannel6Status:=3;
		ELSE
			typChannel6Status:=0;
		END_IF

	(*Channel 7*)
		IF (aDaten[22] AND aDaten[23]) AND (aDaten[6] AND aDaten[7]) THEN
			typChannel7Status:=1;
		ELSIF (aDaten[22] AND aDaten[23]) AND (aDaten[6]=FALSE AND aDaten[7]=FALSE) THEN
			typChannel7Status:=2;
		ELSIF (aDaten[22]=FALSE AND aDaten[23]=FALSE) AND (aDaten[6]=FALSE AND aDaten[7]=FALSE) THEN
			typChannel7Status:=3;
		ELSE
			typChannel7Status:=0;
		END_IF

	(*Channel 8*)
		IF (aDaten[20] AND aDaten[21]) AND (aDaten[4] AND aDaten[5]) THEN
			typChannel8Status:=1;
		ELSIF (aDaten[20] AND aDaten[21]) AND (aDaten[4]=FALSE AND aDaten[5]=FALSE) THEN
			typChannel8Status:=2;
		ELSIF (aDaten[20]=FALSE AND aDaten[21]=FALSE) AND (aDaten[4]=FALSE AND aDaten[5]=FALSE) THEN
			typChannel8Status:=3;
		ELSE
			typChannel8Status:=0;
		END_IF

		(*analog Werte Protokoll 89 bit*)
		IF (aDaten[36] AND aDaten[37]) THEN
			bVoltage.7:=TRUE;
		ELSE
			bVoltage.7:=FALSE;
		END_IF
		IF (aDaten[38] AND aDaten[39]) THEN
			bVoltage.6:=TRUE;
		ELSE
			bVoltage.6:=FALSE;
		END_IF
		IF (aDaten[40] AND aDaten[41]) THEN
			bVoltage.5:=TRUE;
		ELSE
			bVoltage.5:=FALSE;
		END_IF
		IF (aDaten[42] AND aDaten[43]) THEN
			bVoltage.4:=TRUE;
		ELSE
			bVoltage.4:=FALSE;
		END_IF
		IF (aDaten[44] AND aDaten[45]) THEN
			bVoltage.3:=TRUE;
		ELSE
			bVoltage.3:=FALSE;
		END_IF
		IF (aDaten[46] AND aDaten[47]) THEN
			bVoltage.2:=TRUE;
		ELSE
			bVoltage.2:=FALSE;
		END_IF
		IF (aDaten[48] AND aDaten[49]) THEN
			bVoltage.1:=TRUE;
		ELSE
			bVoltage.1:=FALSE;
		END_IF
		IF (aDaten[50] AND aDaten[51]) THEN
			bVoltage.0:=TRUE;
		ELSE
			bVoltage.0:=FALSE;
		END_IF
		IF bVoltage>0 THEN
			rVoltage:=BYTE_TO_REAL(bVoltage)/16+16;
		ELSE
			rVoltage:=0;
		END_IF

		FOR m:=0 TO 7 DO
			IF (aDaten[52+16*m] AND aDaten[53+16*m]) THEN
				auxbyte.7:=TRUE;
			ELSE
				auxbyte.7:=FALSE;
			END_IF
			IF (aDaten[54+16*m] AND aDaten[55+16*m]) THEN
				auxbyte.6:=TRUE;
			ELSE
				auxbyte.6:=FALSE;
			END_IF
			IF (aDaten[56+16*m] AND aDaten[57+16*m]) THEN
				auxbyte.5:=TRUE;
			ELSE
				auxbyte.5:=FALSE;
			END_IF
			IF (aDaten[58+16*m] AND aDaten[59+16*m]) THEN
				auxbyte.4:=TRUE;
			ELSE
				auxbyte.4:=FALSE;
			END_IF
			IF (aDaten[60+16*m] AND aDaten[61+16*m]) THEN
				auxbyte.3:=TRUE;
			ELSE
				auxbyte.3:=FALSE;
			END_IF
			IF (aDaten[62+16*m] AND aDaten[63+16*m]) THEN
				auxbyte.2:=TRUE;
			ELSE
				auxbyte.2:=FALSE;
			END_IF
			IF (aDaten[64+16*m] AND aDaten[65+16*m]) THEN
				auxbyte.1:=TRUE;
			ELSE
				auxbyte.1:=FALSE;
			END_IF
			IF (aDaten[66+16*m] AND aDaten[67+16*m]) THEN
				auxbyte.0:=TRUE;
			ELSE
				auxbyte.0:=FALSE;
			END_IF
			accurrentaux[m]:=auxbyte;
		END_FOR
		rChannel1Current:=BYTE_TO_REAL(accurrentaux[0])/16;
		rChannel2Current:=BYTE_TO_REAL(accurrentaux[1])/16;
		rChannel3Current:=BYTE_TO_REAL(accurrentaux[2])/16;
		rChannel4Current:=BYTE_TO_REAL(accurrentaux[3])/16;
		rChannel5Current:=BYTE_TO_REAL(accurrentaux[4])/16;
		rChannel6Current:=BYTE_TO_REAL(accurrentaux[5])/16;
		rChannel7Current:=BYTE_TO_REAL(accurrentaux[6])/16;
		rChannel8Current:=BYTE_TO_REAL(accurrentaux[7])/16;

		(*indicates wether current or setting values are displayed*)
		xDisplaySettings:=auxProtocolBit5;

		IF auxReset AND xReset THEN
			xReset:=FALSE;
			auxReset:=FALSE;
		END_IF

	3:(*Reset Impuls mit 500ms ausführen*)
		IF xReset  THEN
			xS1_Output:=TRUE;
			TON1(IN:=TRUE , PT:=t#500ms);
			IF ton1.Q THEN
				state:=4;
				TON1(IN:=FALSE);
			END_IF
		ELSE
			state:=5;
			xS1_Output:=FALSE;
		END_IF

	4:(*Pause nach Reset*)
		TON1(IN:=TRUE , PT:=t#300ms);
		xS1_Output:=FALSE;
		IF ton1.Q THEN
			state:=5;
			TON1(IN:=FALSE);
			auxReset:=TRUE;
		END_IF

	5:
	(*Daten anfragen*)

		xS1_Output:=Ausgabe[a];
		aDaten[a+1]:=xS2_Input;
		a:=a+1;
		iauxDisplay:=a;
		auxProtocolBit5:=NOT Ausgabe[22]; (*remember which values should be displayed->current or setting, dependen on bit5*)
		(*IF a>40 THEN*)
		IF a>184 THEN
			state:=0;
			a:=0;
			i:=0;
			go:=FALSE;
			IF 	auxExecute AND xConfigBusy THEN(*schreibauftrag erledigt*)
				xDone:=FALSE;
				auxExecute:=FALSE;
				init:=FALSE;(*damit anschließend nur Daten ausgelesen werden. muss das Feld wieder den Lesecode bekommen*)
			ELSIF auxExecute AND NOT xConfigBusy THEN(*neuer  Schreibauftrag eingetroffen*)
				xConfigBusy:=TRUE;
				xDone:=FALSE;
			ELSE
				IF xConfig THEN
					xDone:=TRUE;
				ELSE
					xDone:=FALSE;
				END_IF
				xConfigBusy:=FALSE;
			END_IF
		ELSE
			;
		END_IF

	END_CASE
ELSE
	xS1_Output:=FALSE;
	state:=0;
	init:=0;
	a:=0;
	i:=0;
	auxReset:=FALSE;
END_IF

END_FUNCTION_BLOCK

// POUs/FB787_1668
FUNCTION_BLOCK FB787_1668
(***********************************************************************************************************	*)
(* Version: 0.8                                    			          														*)
(* Date: 01.07.2013                                   					          							            			*)
(***********************************************************************************************************	*)
(* WAGO Kontakttechnik GmbH Hansastr. 27 32423 Minden(Westf.)									*)
(* Tel. +0049 571/887-0 Fax. +0049 571/887-0															*)
(* Author: VB																								*)
(***********************************************************************************************************	*)
(*Description:	Epsitron electronic fuse	 																*)
(*Historie:																									*)
(*01.07.2013	VB		 Version 0.8 changes according to FW2.00										*)
(*22.10.2012	VB		 Version 0.7 RC																	*)
(***********************************************************************************************************	*)
VAR_INPUT
	xActive							:BOOL;
	xConfig						:BOOL;
	xChannel1Active				:BOOL;
	xChannel2Active				:BOOL;
	xChannel3Active				:BOOL;
	xChannel4Active				:BOOL;
	xChannel5Active				:BOOL;
	xChannel6Active				:BOOL;
	xChannel7Active				:BOOL;
	xChannel8Active				:BOOL;
	xS2_Input						:BOOL;
END_VAR
VAR_OUTPUT
	xDone							:BOOL;
	xConfigBusy					:BOOL;
	typChannel1Status			:typEpsitronStatus;(*0:active,1:Überlast,2:Tripped,3:not_active*)
	typChannel2Status			:typEpsitronStatus;
	typChannel3Status			:typEpsitronStatus;
	typChannel4Status			:typEpsitronStatus;
	typChannel5Status			:typEpsitronStatus;
	typChannel6Status			:typEpsitronStatus;
	typChannel7Status			:typEpsitronStatus;
	typChannel8Status			:typEpsitronStatus;
	xS1_Output					:BOOL;
END_VAR
VAR_IN_OUT
	xReset							:BOOL;
END_VAR
VAR
	a								: INT;
	state							: INT;
	TON1							: TON;
	aDaten						: ARRAY[0..44] OF BOOL;
	i								: INT;
	Ausgabe						: ARRAY[0..44] OF BOOL;
	go								: BOOL;
	init								: BOOL;
	R_TRIG1						: R_TRIG;
	auxExecute					: BOOL;
	auxReset						: BOOL;
END_VAR

IF xActive THEN
	R_TRIG1(CLK:=xConfig);
	IF r_trig1.q THEN
		auxExecute:=TRUE;
	END_IF
	
	CASE state OF
	0:(*ca. 1 Sekunde warten bis der Status abgefragt wird*)

		xS1_Output:=FALSE;
	
		IF NOT init THEN
			Ausgabe[0]:=1;
			Ausgabe[1]:=0;
			Ausgabe[2]:=1;
			Ausgabe[3]:=0;
			Ausgabe[4]:=1;
			Ausgabe[5]:=0;
			Ausgabe[6]:=1;
			Ausgabe[7]:=0;
			Ausgabe[8]:=1;
			Ausgabe[9]:=0;
			Ausgabe[10]:=1;
			Ausgabe[11]:=0;
			Ausgabe[12]:=1;
			Ausgabe[13]:=0;
			Ausgabe[14]:=1;
			Ausgabe[15]:=0;
			Ausgabe[16]:=1;
			Ausgabe[17]:=0;
			Ausgabe[18]:=1;
			Ausgabe[19]:=0;
			Ausgabe[20]:=1;
			Ausgabe[21]:=0;
			Ausgabe[22]:=1;
			Ausgabe[23]:=0;
			Ausgabe[24]:=1;
			Ausgabe[25]:=0;
			Ausgabe[26]:=1;
			Ausgabe[27]:=0;
			Ausgabe[28]:=1;
			Ausgabe[29]:=0;
			Ausgabe[30]:=1;
			Ausgabe[31]:=0;
			Ausgabe[32]:=1;
			Ausgabe[33]:=0;
			Ausgabe[34]:=0;(*1*)
			Ausgabe[35]:=0;
			Ausgabe[36]:=0;
			Ausgabe[37]:=0;
			Ausgabe[38]:=0;
			Ausgabe[39]:=0;
			Ausgabe[40]:=0;
			init:=TRUE;
		END_IF

		IF auxExecute  THEN
			xConfigBusy:=TRUE;
			go:=TRUE;
			Ausgabe[0]:=1;
			Ausgabe[1]:=0;
			IF xChannel8Active THEN
				Ausgabe[2]:=0;
				Ausgabe[3]:=1;
			ELSE
				Ausgabe[2]:=1;
				Ausgabe[3]:=0;
			END_IF
		
			IF xChannel7Active THEN
				Ausgabe[4]:=0;
				Ausgabe[5]:=1;
			ELSE
				Ausgabe[4]:=1;
				Ausgabe[5]:=0;
			END_IF
			IF xChannel6Active THEN
				Ausgabe[6]:=0;
				Ausgabe[7]:=1;
			ELSE
				Ausgabe[6]:=1;
				Ausgabe[7]:=0;
			END_IF
			IF xChannel5Active THEN
				Ausgabe[8]:=0;
				Ausgabe[9]:=1;
			ELSE
				Ausgabe[8]:=1;
				Ausgabe[9]:=0;
			END_IF
			IF xChannel4Active THEN
				Ausgabe[10]:=0;
				Ausgabe[11]:=1;
			ELSE
				Ausgabe[10]:=1;
				Ausgabe[11]:=0;
			END_IF
			IF xChannel3Active THEN
				Ausgabe[12]:=0;
				Ausgabe[13]:=1;
			ELSE
				Ausgabe[12]:=1;
				Ausgabe[13]:=0;
			END_IF
			IF xChannel2Active THEN
				Ausgabe[14]:=0;
				Ausgabe[15]:=1;
			ELSE
				Ausgabe[14]:=1;
				Ausgabe[15]:=0;
			END_IF
			IF xChannel1Active THEN
				Ausgabe[16]:=0;
				Ausgabe[17]:=1;
			ELSE
				Ausgabe[16]:=1;
				Ausgabe[17]:=0;
			END_IF
			IF go THEN
				Ausgabe[18]:=0;
				Ausgabe[19]:=1;
			ELSE
				Ausgabe[18]:=1;
				Ausgabe[19]:=0;
			END_IF
				Ausgabe[20]:=1;
				Ausgabe[21]:=0;
				Ausgabe[22]:=1;
				Ausgabe[23]:=0;
				Ausgabe[24]:=1;
				Ausgabe[25]:=0;
				Ausgabe[26]:=1;
				Ausgabe[27]:=0;
				Ausgabe[28]:=1;
				Ausgabe[29]:=0;
				Ausgabe[30]:=1;
				Ausgabe[31]:=0;
				Ausgabe[32]:=1;
				Ausgabe[33]:=0;
				Ausgabe[34]:=0;(*1*)
				Ausgabe[35]:=0;
				Ausgabe[36]:=0;
				Ausgabe[37]:=0;
				Ausgabe[38]:=0;
				Ausgabe[39]:=0;
				Ausgabe[40]:=0;
				Ausgabe[41]:=0;
				Ausgabe[42]:=0;
				Ausgabe[43]:=0;
				Ausgabe[44]:=0;
		END_IF;

		TON1(IN:=TRUE , PT:=t#1s);
		IF ton1.Q THEN
			state:=3;
			TON1(IN:=FALSE);
		END_IF


		(*Channel 1*)
		IF (aDaten[34] (*AND aDaten[35]*)) AND (aDaten[18] AND aDaten[19]) THEN
			typChannel1Status:=1;
		ELSIF (aDaten[34] (*AND aDaten[35]*)) AND (aDaten[18]=FALSE AND aDaten[19]=FALSE) THEN
			typChannel1Status:=2;
		ELSIF (aDaten[34]=FALSE AND aDaten[35]=FALSE) AND (aDaten[18]=FALSE AND aDaten[19]=FALSE) THEN
			typChannel1Status:=3;
		ELSE
			typChannel1Status:=0;
		END_IF

		(*Channel 2*)
		IF (aDaten[32] AND aDaten[33]) AND (aDaten[16] AND aDaten[17]) THEN
			typChannel2Status:=1;
		ELSIF (aDaten[32] AND aDaten[33]) AND (aDaten[16]=FALSE AND aDaten[17]=FALSE) THEN
			typChannel2Status:=2;
		ELSIF (aDaten[32]=FALSE AND aDaten[33]=FALSE) AND (aDaten[16]=FALSE AND aDaten[17]=FALSE) THEN
			typChannel2Status:=3;
		ELSE
			typChannel2Status:=0;
		END_IF

		(*Channel 3*)
		IF (aDaten[30] AND aDaten[31]) AND (aDaten[14] AND aDaten[15]) THEN
			typChannel3Status:=1;
		ELSIF (aDaten[30] AND aDaten[31]) AND (aDaten[14]=FALSE AND aDaten[15]=FALSE) THEN
			typChannel3Status:=2;
		ELSIF (aDaten[30]=FALSE AND aDaten[31]=FALSE) AND (aDaten[14]=FALSE AND aDaten[15]=FALSE) THEN
			typChannel3Status:=3;
		ELSE
			typChannel3Status:=0;
		END_IF

		(*Channel 4*)
		IF (aDaten[28] AND aDaten[29]) AND (aDaten[12] AND aDaten[13]) THEN
			typChannel4Status:=1;
		ELSIF (aDaten[28] AND aDaten[29]) AND (aDaten[12]=FALSE AND aDaten[13]=FALSE) THEN
			typChannel4Status:=2;
		ELSIF (aDaten[28]=FALSE AND aDaten[29]=FALSE) AND (aDaten[12]=FALSE AND aDaten[13]=FALSE) THEN
			typChannel4Status:=3;
		ELSE
			typChannel4Status:=0;
		END_IF

	(*Channel 5*)
		IF (aDaten[26] AND aDaten[27]) AND (aDaten[10] AND aDaten[11]) THEN
			typChannel5Status:=1;
		ELSIF (aDaten[26] AND aDaten[27]) AND (aDaten[10]=FALSE AND aDaten[11]=FALSE) THEN
			typChannel5Status:=2;
		ELSIF (aDaten[26]=FALSE AND aDaten[27]=FALSE) AND (aDaten[10]=FALSE AND aDaten[11]=FALSE) THEN
			typChannel5Status:=3;
		ELSE
			typChannel5Status:=0;
		END_IF

	(*Channel 6*)
		IF (aDaten[24] AND aDaten[25]) AND (aDaten[8] AND aDaten[9]) THEN
			typChannel6Status:=1;
		ELSIF (aDaten[24] AND aDaten[25]) AND (aDaten[8]=FALSE AND aDaten[9]=FALSE) THEN
			typChannel6Status:=2;
		ELSIF (aDaten[24]=FALSE AND aDaten[25]=FALSE) AND (aDaten[8]=FALSE AND aDaten[9]=FALSE) THEN
			typChannel6Status:=3;
		ELSE
			typChannel6Status:=0;
		END_IF

	(*Channel 7*)
		IF (aDaten[22] AND aDaten[23]) AND (aDaten[6] AND aDaten[7]) THEN
			typChannel7Status:=1;
		ELSIF (aDaten[22] AND aDaten[23]) AND (aDaten[6]=FALSE AND aDaten[7]=FALSE) THEN
			typChannel7Status:=2;
		ELSIF (aDaten[22]=FALSE AND aDaten[23]=FALSE) AND (aDaten[6]=FALSE AND aDaten[7]=FALSE) THEN
			typChannel7Status:=3;
		ELSE
			typChannel7Status:=0;
		END_IF

	(*Channel 8*)
		IF (aDaten[20] AND aDaten[21]) AND (aDaten[4] AND aDaten[5]) THEN
			typChannel8Status:=1;
		ELSIF (aDaten[20] AND aDaten[21]) AND (aDaten[4]=FALSE AND aDaten[5]=FALSE) THEN
			typChannel8Status:=2;
		ELSIF (aDaten[20]=FALSE AND aDaten[21]=FALSE) AND (aDaten[4]=FALSE AND aDaten[5]=FALSE) THEN
			typChannel8Status:=3;
		ELSE
			typChannel8Status:=0;
		END_IF

		IF auxReset AND xReset THEN
			xReset:=FALSE;
			auxReset:=FALSE;
		END_IF

	3:(*Reset Impuls mit 500ms ausführen*)
		IF xReset  THEN
			xS1_Output:=TRUE;
			TON1(IN:=TRUE , PT:=t#500ms);
			IF ton1.Q THEN
				state:=4;
				TON1(IN:=FALSE);
			END_IF
		ELSE
			state:=5;
			xS1_Output:=FALSE;
		END_IF

	4:(*Pause nach Reset*)
		TON1(IN:=TRUE , PT:=t#300ms);
		xS1_Output:=FALSE;
		IF ton1.Q THEN
			state:=5;
			TON1(IN:=FALSE);
			auxReset:=TRUE;
		END_IF

	5:
	(*Daten anfragen*)

		xS1_Output:=Ausgabe[a];
		aDaten[a+1]:=xS2_Input;
		a:=a+1;

		IF a>40 THEN
			state:=0;
			a:=0;
			i:=0;
			go:=FALSE;
			IF 	auxExecute AND xConfigBusy THEN(*schreibauftrag erledigt*)
				xDone:=FALSE;
				auxExecute:=FALSE;
				init:=FALSE;(*damit anschließend nur Daten ausgelesen werden. muss das Feld wieder den Lesecode bekommen*)
			ELSIF auxExecute AND NOT xConfigBusy THEN(*neuer  Schreibauftrag eingetroffen*)
				xConfigBusy:=TRUE;
				xDone:=FALSE;
			ELSE
				IF xConfig THEN
					xDone:=TRUE;
				ELSE
					xDone:=FALSE;
				END_IF
				xConfigBusy:=FALSE;
			END_IF
		ELSE
			;
		END_IF

	END_CASE
ELSE
	xS1_Output:=FALSE;
	state:=0;
	init:=0;
	a:=0;
	i:=0;
	auxReset:=FALSE;
END_IF

END_FUNCTION_BLOCK

// POUs/FB787_1668_ReadCurrent
FUNCTION_BLOCK FB787_1668_ReadCurrent
(***********************************************************************************************************	*)
(* Version: 1.0                                    			          														*)
(* Date: 05.09.2013                                   					          							            			*)
(***********************************************************************************************************	*)
(* WAGO Kontakttechnik GmbH Hansastr. 27 32423 Minden(Westf.)									*)
(* Tel. +0049 571/887-0 Fax. +0049 571/887-0															*)
(* Author: VB																								*)
(***********************************************************************************************************	*)
(*Description:	Epsitron electronic fuse with current overload protection	 							*)
(*Historie:																									*)
(*05.09.2013	VB		 released    																		*)
(***********************************************************************************************************	*)
VAR_INPUT
	xActive							:BOOL;
	xConfig						:BOOL;
	xChannel1Active				:BOOL;
	xChannel2Active				:BOOL;
	xChannel3Active				:BOOL;
	xChannel4Active				:BOOL;
	xChannel5Active				:BOOL;
	xChannel6Active				:BOOL;
	xChannel7Active				:BOOL;
	xChannel8Active				:BOOL;
	xReadSetting					:BOOL;(*0:read current,1:read setting*)
	xS2_Input						:BOOL;
END_VAR
VAR_OUTPUT
	xDone							:BOOL;
	xConfigBusy					:BOOL;
	typChannel1Status			:typEpsitronStatus;(*0:active,1:Überlast,2:Tripped,3:not_active*)
	typChannel2Status			:typEpsitronStatus;
	typChannel3Status			:typEpsitronStatus;
	typChannel4Status			:typEpsitronStatus;
	typChannel5Status			:typEpsitronStatus;
	typChannel6Status			:typEpsitronStatus;
	typChannel7Status			:typEpsitronStatus;
	typChannel8Status			:typEpsitronStatus;
	rVoltage						:REAL;
	rChannel1Current				:REAL;
	rChannel2Current				:REAL;
	rChannel3Current				:REAL;
	rChannel4Current				:REAL;
	rChannel5Current				:REAL;
	rChannel6Current				:REAL;
	rChannel7Current				:REAL;
	rChannel8Current				:REAL;
	iauxDisplay					:INT;
	xDisplaySettings				:BOOL;(*0:Channel value is current, 1:Channel value is setting*)
	xS1_Output					:BOOL;
END_VAR
VAR_IN_OUT
	xReset							:BOOL;
END_VAR
VAR
	a								: INT;
	state							: INT;
	TON1							: TON;
	aDaten						: ARRAY[0..188] OF BOOL;
	i								: INT;
	Ausgabe						: ARRAY[0..188] OF BOOL;
	go								: BOOL;
	init								: BOOL;
	R_TRIG1						: R_TRIG;
	auxExecute					: BOOL;
	auxReset						: BOOL;
	k								: INT;
	m								: INT;
	auxbyte						: BYTE;
	accurrentaux					: ARRAY[0..7]OF BYTE;
	bVoltage						: BYTE;
	auxProtocolBit5				: BOOL;
END_VAR

IF xActive THEN
	R_TRIG1(CLK:=xConfig);
	IF r_trig1.q THEN
		auxExecute:=TRUE;
	END_IF
	
	CASE state OF
	0:(*ca. 1 Sekunde warten bis der Status abgefragt wird*)

		xS1_Output:=FALSE;

		IF xReadSetting THEN
			Ausgabe[22]:=0;(*Bit 5->true*)
			Ausgabe[23]:=1;
		ELSE
			Ausgabe[22]:=1;
			Ausgabe[23]:=0;
		END_IF

		IF NOT init THEN
			FOR k:=0 TO 89 DO
				Ausgabe[2*k]:=1;
				Ausgabe[2*k+1]:=0;
			END_FOR
			FOR k:=0 TO 8 DO
				Ausgabe[178+k]:=0;
			END_FOR
			(*Protokoll 89 Bit*)
			Ausgabe[20]:=0;(*bit 6->true*)
			Ausgabe[21]:=1;

			IF xReadSetting THEN
				Ausgabe[22]:=0;(*Bit 5->true*)
				Ausgabe[23]:=1;
			ELSE
				Ausgabe[22]:=1;
				Ausgabe[23]:=0;
			END_IF

			init:=TRUE;
		END_IF

		IF auxExecute  THEN
			xConfigBusy:=TRUE;
			go:=TRUE;
			Ausgabe[0]:=1;
			Ausgabe[1]:=0;
			IF xChannel8Active THEN
				Ausgabe[2]:=0;
				Ausgabe[3]:=1;
			ELSE
				Ausgabe[2]:=1;
				Ausgabe[3]:=0;
			END_IF
		
			IF xChannel7Active THEN
				Ausgabe[4]:=0;
				Ausgabe[5]:=1;
			ELSE
				Ausgabe[4]:=1;
				Ausgabe[5]:=0;
			END_IF
			IF xChannel6Active THEN
				Ausgabe[6]:=0;
				Ausgabe[7]:=1;
			ELSE
				Ausgabe[6]:=1;
				Ausgabe[7]:=0;
			END_IF
			IF xChannel5Active THEN
				Ausgabe[8]:=0;
				Ausgabe[9]:=1;
			ELSE
				Ausgabe[8]:=1;
				Ausgabe[9]:=0;
			END_IF
			IF xChannel4Active THEN
				Ausgabe[10]:=0;
				Ausgabe[11]:=1;
			ELSE
				Ausgabe[10]:=1;
				Ausgabe[11]:=0;
			END_IF
			IF xChannel3Active THEN
				Ausgabe[12]:=0;
				Ausgabe[13]:=1;
			ELSE
				Ausgabe[12]:=1;
				Ausgabe[13]:=0;
			END_IF
			IF xChannel2Active THEN
				Ausgabe[14]:=0;
				Ausgabe[15]:=1;
			ELSE
				Ausgabe[14]:=1;
				Ausgabe[15]:=0;
			END_IF
			IF xChannel1Active THEN
				Ausgabe[16]:=0;
				Ausgabe[17]:=1;
			ELSE
				Ausgabe[16]:=1;
				Ausgabe[17]:=0;
			END_IF
			IF go THEN
				Ausgabe[18]:=0;
				Ausgabe[19]:=1;
			ELSE
				Ausgabe[18]:=1;
				Ausgabe[19]:=0;
			END_IF

			(*Protokoll 89 Bit*)
			Ausgabe[20]:=0;
			Ausgabe[21]:=1;
			IF xReadSetting THEN
				Ausgabe[22]:=0;(*Bit 5->true*)
				Ausgabe[23]:=1;
			ELSE
				Ausgabe[22]:=1;
				Ausgabe[23]:=0;
			END_IF

				FOR k:=0 TO 79 DO
					Ausgabe[24+2*k]:=1;
					Ausgabe[25+2*k]:=0;
				END_FOR

				Ausgabe[178]:=0;
				Ausgabe[179]:=0;
				Ausgabe[180]:=0;
				Ausgabe[181]:=0;
				Ausgabe[182]:=0;
				Ausgabe[183]:=0;
				Ausgabe[184]:=0;
				Ausgabe[185]:=0;
				Ausgabe[186]:=0;
				Ausgabe[187]:=0;
				Ausgabe[188]:=0;

		END_IF;

		TON1(IN:=TRUE , PT:=t#1s);
		IF ton1.Q THEN
			state:=3;
			TON1(IN:=FALSE);
		END_IF


		(*Channel 1*)
		IF (aDaten[34] (*AND aDaten[35]*)) AND (aDaten[18] AND aDaten[19]) THEN
			typChannel1Status:=1;
		ELSIF (aDaten[34] (*AND aDaten[35]*)) AND (aDaten[18]=FALSE AND aDaten[19]=FALSE) THEN
			typChannel1Status:=2;
		ELSIF (aDaten[34]=FALSE AND aDaten[35]=FALSE) AND (aDaten[18]=FALSE AND aDaten[19]=FALSE) THEN
			typChannel1Status:=3;
		ELSE
			typChannel1Status:=0;
		END_IF

		(*Channel 2*)
		IF (aDaten[32] AND aDaten[33]) AND (aDaten[16] AND aDaten[17]) THEN
			typChannel2Status:=1;
		ELSIF (aDaten[32] AND aDaten[33]) AND (aDaten[16]=FALSE AND aDaten[17]=FALSE) THEN
			typChannel2Status:=2;
		ELSIF (aDaten[32]=FALSE AND aDaten[33]=FALSE) AND (aDaten[16]=FALSE AND aDaten[17]=FALSE) THEN
			typChannel2Status:=3;
		ELSE
			typChannel2Status:=0;
		END_IF

		(*Channel 3*)
		IF (aDaten[30] AND aDaten[31]) AND (aDaten[14] AND aDaten[15]) THEN
			typChannel3Status:=1;
		ELSIF (aDaten[30] AND aDaten[31]) AND (aDaten[14]=FALSE AND aDaten[15]=FALSE) THEN
			typChannel3Status:=2;
		ELSIF (aDaten[30]=FALSE AND aDaten[31]=FALSE) AND (aDaten[14]=FALSE AND aDaten[15]=FALSE) THEN
			typChannel3Status:=3;
		ELSE
			typChannel3Status:=0;
		END_IF

		(*Channel 4*)
		IF (aDaten[28] AND aDaten[29]) AND (aDaten[12] AND aDaten[13]) THEN
			typChannel4Status:=1;
		ELSIF (aDaten[28] AND aDaten[29]) AND (aDaten[12]=FALSE AND aDaten[13]=FALSE) THEN
			typChannel4Status:=2;
		ELSIF (aDaten[28]=FALSE AND aDaten[29]=FALSE) AND (aDaten[12]=FALSE AND aDaten[13]=FALSE) THEN
			typChannel4Status:=3;
		ELSE
			typChannel4Status:=0;
		END_IF

	(*Channel 5*)
		IF (aDaten[26] AND aDaten[27]) AND (aDaten[10] AND aDaten[11]) THEN
			typChannel5Status:=1;
		ELSIF (aDaten[26] AND aDaten[27]) AND (aDaten[10]=FALSE AND aDaten[11]=FALSE) THEN
			typChannel5Status:=2;
		ELSIF (aDaten[26]=FALSE AND aDaten[27]=FALSE) AND (aDaten[10]=FALSE AND aDaten[11]=FALSE) THEN
			typChannel5Status:=3;
		ELSE
			typChannel5Status:=0;
		END_IF

	(*Channel 6*)
		IF (aDaten[24] AND aDaten[25]) AND (aDaten[8] AND aDaten[9]) THEN
			typChannel6Status:=1;
		ELSIF (aDaten[24] AND aDaten[25]) AND (aDaten[8]=FALSE AND aDaten[9]=FALSE) THEN
			typChannel6Status:=2;
		ELSIF (aDaten[24]=FALSE AND aDaten[25]=FALSE) AND (aDaten[8]=FALSE AND aDaten[9]=FALSE) THEN
			typChannel6Status:=3;
		ELSE
			typChannel6Status:=0;
		END_IF

	(*Channel 7*)
		IF (aDaten[22] AND aDaten[23]) AND (aDaten[6] AND aDaten[7]) THEN
			typChannel7Status:=1;
		ELSIF (aDaten[22] AND aDaten[23]) AND (aDaten[6]=FALSE AND aDaten[7]=FALSE) THEN
			typChannel7Status:=2;
		ELSIF (aDaten[22]=FALSE AND aDaten[23]=FALSE) AND (aDaten[6]=FALSE AND aDaten[7]=FALSE) THEN
			typChannel7Status:=3;
		ELSE
			typChannel7Status:=0;
		END_IF

	(*Channel 8*)
		IF (aDaten[20] AND aDaten[21]) AND (aDaten[4] AND aDaten[5]) THEN
			typChannel8Status:=1;
		ELSIF (aDaten[20] AND aDaten[21]) AND (aDaten[4]=FALSE AND aDaten[5]=FALSE) THEN
			typChannel8Status:=2;
		ELSIF (aDaten[20]=FALSE AND aDaten[21]=FALSE) AND (aDaten[4]=FALSE AND aDaten[5]=FALSE) THEN
			typChannel8Status:=3;
		ELSE
			typChannel8Status:=0;
		END_IF

		(*analog Werte Protokoll 89 bit*)
		IF (aDaten[36] AND aDaten[37]) THEN
			bVoltage.7:=TRUE;
		ELSE
			bVoltage.7:=FALSE;
		END_IF
		IF (aDaten[38] AND aDaten[39]) THEN
			bVoltage.6:=TRUE;
		ELSE
			bVoltage.6:=FALSE;
		END_IF
		IF (aDaten[40] AND aDaten[41]) THEN
			bVoltage.5:=TRUE;
		ELSE
			bVoltage.5:=FALSE;
		END_IF
		IF (aDaten[42] AND aDaten[43]) THEN
			bVoltage.4:=TRUE;
		ELSE
			bVoltage.4:=FALSE;
		END_IF
		IF (aDaten[44] AND aDaten[45]) THEN
			bVoltage.3:=TRUE;
		ELSE
			bVoltage.3:=FALSE;
		END_IF
		IF (aDaten[46] AND aDaten[47]) THEN
			bVoltage.2:=TRUE;
		ELSE
			bVoltage.2:=FALSE;
		END_IF
		IF (aDaten[48] AND aDaten[49]) THEN
			bVoltage.1:=TRUE;
		ELSE
			bVoltage.1:=FALSE;
		END_IF
		IF (aDaten[50] AND aDaten[51]) THEN
			bVoltage.0:=TRUE;
		ELSE
			bVoltage.0:=FALSE;
		END_IF
		IF bVoltage>0 THEN
			rVoltage:=BYTE_TO_REAL(bVoltage)/16+16;
		ELSE
			rVoltage:=0;
		END_IF


		FOR m:=0 TO 7 DO
			IF (aDaten[52+16*m] AND aDaten[53+16*m]) THEN
				auxbyte.7:=TRUE;
			ELSE
				auxbyte.7:=FALSE;
			END_IF
			IF (aDaten[54+16*m] AND aDaten[55+16*m]) THEN
				auxbyte.6:=TRUE;
			ELSE
				auxbyte.6:=FALSE;
			END_IF
			IF (aDaten[56+16*m] AND aDaten[57+16*m]) THEN
				auxbyte.5:=TRUE;
			ELSE
				auxbyte.5:=FALSE;
			END_IF
			IF (aDaten[58+16*m] AND aDaten[59+16*m]) THEN
				auxbyte.4:=TRUE;
			ELSE
				auxbyte.4:=FALSE;
			END_IF
			IF (aDaten[60+16*m] AND aDaten[61+16*m]) THEN
				auxbyte.3:=TRUE;
			ELSE
				auxbyte.3:=FALSE;
			END_IF
			IF (aDaten[62+16*m] AND aDaten[63+16*m]) THEN
				auxbyte.2:=TRUE;
			ELSE
				auxbyte.2:=FALSE;
			END_IF
			IF (aDaten[64+16*m] AND aDaten[65+16*m]) THEN
				auxbyte.1:=TRUE;
			ELSE
				auxbyte.1:=FALSE;
			END_IF
			IF (aDaten[66+16*m] AND aDaten[67+16*m]) THEN
				auxbyte.0:=TRUE;
			ELSE
				auxbyte.0:=FALSE;
			END_IF
			accurrentaux[m]:=auxbyte;
		END_FOR
		rChannel1Current:=BYTE_TO_REAL(accurrentaux[0])/16;
		rChannel2Current:=BYTE_TO_REAL(accurrentaux[1])/16;
		rChannel3Current:=BYTE_TO_REAL(accurrentaux[2])/16;
		rChannel4Current:=BYTE_TO_REAL(accurrentaux[3])/16;
		rChannel5Current:=BYTE_TO_REAL(accurrentaux[4])/16;
		rChannel6Current:=BYTE_TO_REAL(accurrentaux[5])/16;
		rChannel7Current:=BYTE_TO_REAL(accurrentaux[6])/16;
		rChannel8Current:=BYTE_TO_REAL(accurrentaux[7])/16;

		(*indicates wether current or setting values are displayed*)
		xDisplaySettings:=auxProtocolBit5;


		IF auxReset AND xReset THEN
			xReset:=FALSE;
			auxReset:=FALSE;
		END_IF

	3:(*Reset Impuls mit 500ms ausführen*)
		IF xReset  THEN
			xS1_Output:=TRUE;
			TON1(IN:=TRUE , PT:=t#500ms);
			IF ton1.Q THEN
				state:=4;
				TON1(IN:=FALSE);
			END_IF
		ELSE
			state:=5;
			xS1_Output:=FALSE;
		END_IF

	4:(*Pause nach Reset*)
		TON1(IN:=TRUE , PT:=t#300ms);
		xS1_Output:=FALSE;
		IF ton1.Q THEN
			state:=5;
			TON1(IN:=FALSE);
			auxReset:=TRUE;
		END_IF

	5:
	(*Daten anfragen*)

		xS1_Output:=Ausgabe[a];
		aDaten[a+1]:=xS2_Input;
		a:=a+1;
		iauxDisplay:=a;
		auxProtocolBit5:=NOT Ausgabe[22]; (*remember which values should be displayed->current or setting, dependen on bit5*)
		(*IF a>40 THEN*)
		IF a>184 THEN
			state:=0;
			a:=0;
			i:=0;
			go:=FALSE;
			IF 	auxExecute AND xConfigBusy THEN(*schreibauftrag erledigt*)
				xDone:=FALSE;
				auxExecute:=FALSE;
				init:=FALSE;(*damit anschließend nur Daten ausgelesen werden. muss das Feld wieder den Lesecode bekommen*)
			ELSIF auxExecute AND NOT xConfigBusy THEN(*neuer  Schreibauftrag eingetroffen*)
				xConfigBusy:=TRUE;
				xDone:=FALSE;
			ELSE
				IF xConfig THEN
					xDone:=TRUE;
				ELSE
					xDone:=FALSE;
				END_IF
				xConfigBusy:=FALSE;
			END_IF
		ELSE
			;
		END_IF

	END_CASE
ELSE
	xS1_Output:=FALSE;
	state:=0;
	init:=0;
	a:=0;
	i:=0;
	auxReset:=FALSE;
END_IF

END_FUNCTION_BLOCK

// POUs/FC787_Version
FUNCTION FC787_Version : WORD
(*Version 1.3

  date    	  | release			  | author  |
------------------+---------------------+------------------------------------------------------------------------------------------------------- 
 04.11.14	  |	1.3			 	  | VB          | FB787_1675  comment wStatus added 
 05.09.13	  |	1.2			 	  | VB          | 89-Bit Support for FB787_166x(ReadCurrent),  
 01.07.13	  |	1.1			 	  | VB          | Changes according to FW 2.0 ->FB787_166x 
 13.05.13	  |	0.9			 	  | VB          | New Function block FB787_1675 
 19.04.13	  |	0.8			 	  | VB          | Output FB787_166x enum changed
 23.10.12	  |	0.7			 	  | VB          | Improvement output FB787_166x
 04.10.12	  |	0.6			 	  | VB          | New Function blocks FB787_166x for Epsitron Classic Power
 01.03.10	  |	0.5			 	  | VB          | Update FB78787x to protocol description 1.2
 01.10.09	  |	0.4			 	  | VB          | Improvement output xValid
 02.09.09	  |	0.3			 	  | VB          | Bugfix 787-85x
 02.07.09	  | 	0.2			 	  | JK          | Extension  to read the device parameters.
 			  | 	0.1			 	  | JB          |  Init version
----------------+-----------------------+------------------------------------------------------------------------------------------------------------*)


VAR_INPUT
END_VAR
VAR
	bMajor : BYTE := 16#01; (* Major version number *)
	bMinor : BYTE := 16#03; (* Minor version number *)
END_VAR

FC787_Version := SHL(BYTE_TO_WORD(bMajor), 4) OR bMinor;

END_FUNCTION
